PROGRAM MAIN
VAR
	// Close hand signal from output of C6032
	bServoClosedSignal AT %I*	:	BOOL;
	

	// PWM Controls
	iPWMOutput AT %Q*			:	UINT;
	iPWMPeriod AT %Q*			:	UINT;

END_VAR

iPWMPeriod := 10000;
IF bServoClosedSignal THEN
	iPWMOutput := 9000;
ELSE
	iPWMOutput := 3300;
END_IF

END_PROGRAM

(* stored: Version 1.1.0.1, ProductVersion 3.1.4024.12
   POU MAIN: Id {82899c5e-3dbe-4415-8592-db38cca79af8}, SpecialFunc None *)
